PROGRAM MAIN
VAR
	_station001	:	Station001;
	_station002	:	Station002;
END_VAR

EXAMPLES_PRG();
MANIPULATOR();
_station001._sequence.DeactivateDeveloperChecks();

_station001.Run();
_station002.Run();

END_PROGRAM

(* stored: Version 1.1.0.1
   POU MAIN: Id {a7bd41fd-8dbf-4e6f-8b13-73b5ce6425f6}, SpecialFunc None *)
